PROGRAM PRG_FB_AxisServoCA_PreTest
VAR
	bFirstCycle : BOOL := TRUE;
	
	AxesGroupRef		: AXES_GROUP_REF;
	stAxisRef			: AXIS_REF;
	
	fbAxisCA1			: FB_AxisServoCA;
	fbAxisCA2			: FB_AxisServoCA;
	
	fbAddAxisToGroup 	: MC_AddAxisToGroup;
	fbGroupEnable		: MC_GroupEnable;
	fbGroupReset		: MC_GroupReset;
	
	fbReadGroupStatus	: MC_GroupReadStatus;
	fbReadGroupError	: MC_GroupReadError;
	
	fbMcMoveAbsCA 		: MC_MoveAbsoluteCA;
	
	iState : INT;
	
	bAdd		: BOOL;
	bReset		: BOOL;
	bInit 		: BOOL;
	bDeinit 	: BOOL;
	bHome		: BOOL;
	bMoveAbsCA1 : BOOL;
	bMoveAbsCA2 : BOOL;
	bStop 		: BOOL;
	bHalt: BOOL;
	
	rHomePosition 		: REAL := 0.0;
	rTargetPositionCA1 	: REAL;
	rTargetPositionCA2 	: REAL;
	
	bAdded : BOOL;
	
	lrOverride: LREAL;
	lrVelocity: LREAL;
	lrAcceleration: LREAL;
	lrDeceleration: LREAL;
	lrJerk: LREAL;
	lrJogVelocity: LREAL;
	lrJogAcceleration: LREAL;
	lrJogDeceleration: LREAL;
	lrJogJerk: LREAL;
	lrStopDeceleration: LREAL;
	lrStopJerk: LREAL;
END_VAR

IF bFirstCycle THEN
	bFirstCycle := FALSE;
	
	lrOverride 			:= 100.0;
	lrVelocity 			:= 50.0;
	lrAcceleration		:= 150.0;
	lrDeceleration		:= 150.0;
	lrJerk				:= 150.0;
	
	lrJogVelocity 		:= 25.0;
	lrJogAcceleration	:= 250.0;
	lrJogDeceleration	:= 250.0;
	lrJogJerk			:= 250.0;
	
	lrStopDeceleration	:= 250.0;
	lrStopJerk			:= 250.0;
	
	fbAxisCA1.Override 			:= lrOverride;
	fbAxisCA1.Velocity 			:= lrVelocity;
	fbAxisCA1.Acceleration 		:= lrAcceleration;
	fbAxisCA1.Deceleration 		:= lrDeceleration;
	fbAxisCA1.Jerk 				:= lrJerk;
	fbAxisCA1.StopDeceleration 	:= lrStopDeceleration;
	fbAxisCA1.StopJerk			:= lrStopJerk;
	
	fbAxisCA2.Override 			:= lrOverride;
	fbAxisCA2.Velocity 			:= lrVelocity;
	fbAxisCA2.Acceleration 		:= lrAcceleration;
	fbAxisCA2.Deceleration 		:= lrDeceleration;
	fbAxisCA2.Jerk 				:= lrJerk;
	fbAxisCA2.StopDeceleration 	:= lrStopDeceleration;
	fbAxisCA2.StopJerk			:= lrStopJerk;
	
END_IF

IF bStop THEN
	bStop := FALSE;
	iState := 100;
ELSIF bHalt THEN
	bHalt := FALSE;
	iState := 110;
END_IF

fbReadGroupStatus( AxesGroup := AxesGroupRef, Enable := TRUE);
fbReadGroupError( AxesGroup := AxesGroupRef, Enable := TRUE);

CASE iState OF
	0:
		IF bAdd THEN
			bAdded := FALSE;
			bAdd := FALSE;
			iState := 10;
		ELSIF bReset THEN
			bReset := FALSE;
			iState := 5;
			
		ELSIF bInit THEN
			bInit := FALSE;
			iState := 50;
			
		ELSIF bDeinit THEN
			bDeinit := FALSE;
			iState := 60;
			
		ELSIF bHome THEN
			bHome := FALSE;
			iState := 70;
		
		ELSIF bMoveAbsCA1 THEN
			bMoveAbsCA1 := FALSE;
			iState := 80;
			
		ELSIF bMoveAbsCA2 THEN
			bMoveAbsCA2 := FALSE;
			iState := 90;
			
		END_IF
	5:
		fbGroupReset( AxesGroup := AxesGroupRef, Execute := TRUE);
		
		IF fbGroupReset.Done THEN
			fbGroupReset( AxesGroup := AxesGroupRef, Execute := FALSE);
			iState := 0;
		END_IF
		
	10:
		stAxisRef := fbAxisCA1.AxisRef;
		fbAddAxisToGroup( 	AxesGroup := AxesGroupRef,
							Axis := stAxisRef,
							Execute := TRUE,
							IdentInGroup := UDINT_TO_IDENTINGROUP(1));
							
		IF fbAddAxisToGroup.Done THEN
			iState := 20;
		END_IF
		
	20:
		fbAddAxisToGroup( AxesGroup := AxesGroupRef , Axis := stAxisRef, Execute := FALSE);
		
		IF NOT fbAddAxisToGroup.Busy THEN
			iState := 30;
		END_IF
		
	30:
		stAxisRef := fbAxisCA2.AxisRef;
		fbAddAxisToGroup( 	AxesGroup := AxesGroupRef,
							Axis := stAxisRef,
							Execute := TRUE,
							IdentInGroup := UDINT_TO_IDENTINGROUP(2));
							
		IF fbAddAxisToGroup.Done THEN
			iState := 40;
		END_IF
		
	40:
		fbAddAxisToGroup( AxesGroup := AxesGroupRef , Axis := stAxisRef, Execute := FALSE);
		
		IF NOT fbAddAxisToGroup.Busy THEN
			bAdded := TRUE;
			iState := 45;
		END_IF
		
	45:
		
		fbGroupEnable( AxesGroup := AxesGroupRef, Execute := TRUE);
		
		IF fbGroupEnable.Done THEN
			fbGroupEnable( AxesGroup := AxesGroupRef, Execute := FALSE);
			iState := 0;
		END_IF
		
	50:
		fbAxisCA1.MR_Init();
		IF fbAxisCA1.State = E_AxisState.AXIS_READY THEN
			iState := 55;
		END_IF
		
	55:
	
		fbAxisCA2.MR_Init();
		IF fbAxisCA2.State = E_AxisState.AXIS_READY THEN
			iState := 0;
		END_IF
		
	60:
		fbAxisCA1.MR_Deinit();
		fbAxisCA2.MR_Deinit();
		
		IF NOT fbAxisCA1.PowerOn AND NOT fbAxisCA2.PowerOn THEN
			iState := 0;
		END_IF
		
	70:
		fbAxisCA1.MR_Home(0.0);
		
		IF fbAxisCA1.IsHomed THEN
			iState := 75;
		END_IF
		
	75:
		fbAxisCA2.MR_Home(3000.0);
		
		IF fbAxisCA2.IsHomed THEN
			iState := 0;
		END_IF
		
	80:
		fbAxisCA1.MR_MoveAbsolute(rTargetPositionCA1);
		
		IF fbAxisCA1.InPosition THEN
			iState := 0;
		END_IF
		
	90:
		fbAxisCA2.MR_MoveAbsolute(rTargetPositionCA2);
		
		IF fbAxisCA2.InPosition THEN
			iState := 0;
		END_IF
		
	100:
		fbAxisCA1.MR_Stop();
		fbAxisCA2.MR_Stop();

		IF fbAxisCA1.Stopped AND fbAxisCA2.Stopped THEN
			iState := 0;
		END_IF;	
	110:
		fbAxisCA1.MR_Halt();
		fbAxisCA2.MR_Halt();
		
		IF fbAxisCA1.Halted AND fbAxisCA2.Halted THEN
			iState := 0;
		END_IF
		
END_CASE

fbAxisCA1();
fbAxisCA2();

END_PROGRAM

(* stored: Version 1.1.0.1, ProductVersion 3.1.4024.9
   POU PRG_FB_AxisServoCA_PreTest: Id {cebed05c-6946-4e14-83fb-fcfa8617100b}, SpecialFunc None *)
